// TIA Portal V18 export
VAR_GLOBAL   // PLC tag table "HMI"
   "HMI - AntiCrash UltraSonic ByPass" AT %M801.0 : Bool;
   "HMI - Auto Floor" AT %M801.3 : Bool;
   "HMI - Fire Siren Acitve/Passive" AT %M801.2 : Bool;
   "HMI - Floor Auto Mode" AT %M800.7 : Bool;
   "HMI - Int Light Button" AT %M801.1 : Bool;
   "HMI - Lamp Test Button" AT %M800.6 : Bool;
   "HMI Power output" AT %Q10.0 : Bool;   // R36 -
   "HMI R1 - Plane Door Light" AT %M800.1 : Bool;
   "HMI R2 - Plane Door Light" AT %M800.2 : Bool;
   "HMI R3 - Drive Unit Light" AT %M800.3 : Bool;
   "HMI R4 - Cabin Front Light" AT %M800.4 : Bool;
   "HMI R6 - SafetyEdge Light" AT %M800.5 : Bool;
   "HMI SafetyEdge Bypass" AT %M800.0 : Bool;
END_VAR
